{attribute 'GeneratedUsingTerminal: EK1960-0000-0019'}
{attribute addProperty BoxType "EK1960-0000-0019"}
{attribute addProperty Id "AdsAddrAT %I*.TcoAmsAddr0StateAT %I*UINT2"}
{attribute addProperty CRC "2493615966"}
{attribute addProperty Size "2"}
TYPE InfoData_94A18F5E EXTENDS InputBase_8311D824 :
STRUCT
	{attribute addProperty Name "AdsAddr"}
	AdsAddr AT %I* : .TcoAmsAddr;
	{attribute addProperty Name "State"}
	State AT %I* : UINT;
END_STRUCT
END_TYPE

(* stored: Version 1.2.0.0, ProductVersion 3.1.4024.9
   DUT InfoData_94A18F5E: Id {cb31618e-4cb9-4a03-9dc7-26dc60bbefff} *)
